ABB RobotStudio station: RobotStudio-Project-01.rspag

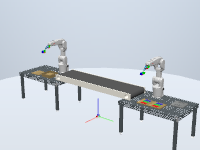
--- station ---
Station RobotStudio-Project-01 (saved by RobotStudio 20.4.9280.0)
Controller Controller1, task T_ROB2: task frame (RAPID world) sits at (-301.82, 1547.77, 837.1) mm in the station
Controller Controller1, task T_ROB1: task frame (RAPID world) sits at (-301.82, 1547.77, 837.1) mm in the station
Controller Controller1
  mechanical unit ROB_1: IRB1200_5_90_STD_03_1, 6 joints, base frame (0, 0, 0) mm
  mechanical unit ROB_2: IRB1200_5_90_STD_03_2, 6 joints, base frame (0, -3095.03, 0) mm
Layout (positions relative to the parent item):
  - WALL [part]
  - CONV_BELT [part] at (300.5, 959.08, 865.68) mm, rotated rx 90 ry 0 rz -90 deg
  - TABLE_1 [part] at (-6.2, -768.26, 800) mm, rotated rx 90 ry 0 rz 180 deg
  - TABLE_2 [part] at (-5.7, -4268.26, 800) mm, rotated rx 90 ry 0 rz 180 deg
  - TAB_1_ALL [part] at (184.19, 1489.88, 847.1) mm
  - TAB_2_ALL [part] at (184.19, 1790.38, 847.1) mm
  - TAB_3_HOME [part] at (-149.02, 2188.84, 854.6) mm
  - BOX [part] at (204.09, -1572.68, 882.1) mm, rotated rx 180 ry 0 rz 180 deg
  - BOX_COVER_ONBOX [part] at (204.09, -1572.68, 882.1) mm, rotated rx 180 ry 0 rz 180 deg
  - BOX_COVER_HOME [part] at (209.09, -2017.68, 802.1) mm, rotated rx 180 ry 0 rz 180 deg
  - TAB_1_POS_1 [part] at (184.19, 1489.88, 847.1) mm
  - TAB_1_POS_3 [part] at (184.19, 1489.88, 847.1) mm
  - TAB_1_POS_2 [part] at (184.19, 1489.88, 847.1) mm
  - TAB_2_POS_1 [part] at (184.19, 1790.38, 847.1) mm
  - TAB_2_POS_3 [part] at (184.19, 1790.38, 847.1) mm
  - TAB_2_POS_2 [part] at (184.19, 1790.38, 847.1) mm
  - TAB_3_CONV_1 [part] at (1.48, 950, 994.6) mm
  - TAB_3_CONV_2 [part] at (1.48, -975, 994.6) mm
  - TAB_3_INBOX [part] at (191.48, -1570.66, 884.6) mm
  - TAB_3_CONV_1_POS_1 [part] at (1.48, 950, 994.6) mm
  - TAB_3_CONV_1_POS_2 [part] at (1.48, 950, 994.6) mm
  - IRB1200_5_90_STD_03_1 [mechanism, from Robots\IRB1200_5_90_STD_03.rslib] at (-301.82, 1547.77, 837.1) mm; joint values [0, 0, 0, 0, 0.5236, 0] (rad or m)
  - IRB1200_5_90_STD_03_2 [mechanism, from Robots\IRB1200_5_90_STD_03.rslib] at (-301.82, -1547.27, 837.1) mm; joint values [0, 0, 0, 0, 0.5236, 0] (rad or m)
  - smc_gripper_1 [mechanism, from .rslib\smc_gripper.rslib] at (220.19, 1547.77, 1685.2) mm, rotated rx 180 ry 60 rz 180 deg
  - smc_gripper_2 [mechanism, from .rslib\smc_gripper.rslib] at (220.19, -1547.27, 1685.2) mm, rotated rx 180 ry 60 rz 180 deg
  - Detacher_T3_1 [smart component, from Components\Detacher.rslib]
      properties: Child=TAB_3_HOME; KeepPosition=true
  - Attacher_T3_1 [smart component, from Components\Attacher.rslib]
      properties: Parent=smc_gripper_1; Flange=0; Child=TAB_3_HOME; Mount=false; Offset=[0 0 0]; Orientation=[0 0 0]
  - Attacher_T1_P1 [smart component, from Components\Attacher.rslib]
      properties: Parent=smc_gripper_1; Flange=0; Child=TAB_1_POS_1; Mount=false; Offset=[0 0 0]; Orientation=[0 0 0]
  - Detacher_T1_P1 [smart component, from Components\Detacher.rslib]
      properties: Child=TAB_1_POS_1; KeepPosition=true
  - Attacher_T2_P1 [smart component, from Components\Attacher.rslib]
      properties: Parent=smc_gripper_1; Flange=0; Child=TAB_2_POS_1; Mount=false; Offset=[0 0 0]; Orientation=[0 0 0]
  - Detacher_T2_P1 [smart component, from Components\Detacher.rslib]
      properties: Child=TAB_2_POS_1; KeepPosition=true
  - Attacher_T1_P2 [smart component, from Components\Attacher.rslib]
      properties: Parent=smc_gripper_1; Flange=0; Child=TAB_1_POS_2; Mount=false; Offset=[0 0 0]; Orientation=[0 0 0]
  - Detacher_T1_P2 [smart component, from Components\Detacher.rslib]
      properties: Child=TAB_1_POS_2; KeepPosition=true
  - Attacher_T2_P2 [smart component, from Components\Attacher.rslib]
      properties: Parent=smc_gripper_1; Flange=0; Child=TAB_2_POS_2; Mount=false; Offset=[0 0 0]; Orientation=[0 0 0]
  - Detacher_T2_P2 [smart component, from Components\Detacher.rslib]
      properties: Child=TAB_2_POS_2; KeepPosition=true
  - Attacher_T1_P3 [smart component, from Components\Attacher.rslib]
      properties: Parent=smc_gripper_1; Flange=0; Child=TAB_1_POS_3; Mount=false; Offset=[0 0 0]; Orientation=[0 0 0]
  - Detacher_T1_P3 [smart component, from Components\Detacher.rslib]
      properties: Child=TAB_1_POS_3; KeepPosition=true
  - Attacher_T2_P3 [smart component, from Components\Attacher.rslib]
      properties: Parent=smc_gripper_1; Flange=0; Child=TAB_2_POS_3; Mount=false; Offset=[0 0 0]; Orientation=[0 0 0]
  - Detacher_T2_P3 [smart component, from Components\Detacher.rslib]
      properties: Child=TAB_2_POS_3; KeepPosition=true
  - Attacher_T3_2 [smart component, from Components\Attacher.rslib]
      properties: Parent=smc_gripper_2; Flange=0; Child=TAB_3_HOME; Mount=false; Offset=[0 0 0]; Orientation=[0 0 0]
  - Detacher_T3_2 [smart component, from Components\Detacher.rslib]
      properties: Child=TAB_3_HOME; KeepPosition=true
  - Attacher_BC [smart component, from Components\Attacher.rslib]
      properties: Parent=smc_gripper_2; Flange=0; Child=BOX_COVER_HOME; Mount=false; Offset=[0 0 0]; Orientation=[0 0 0]
  - Detacher_BC [smart component, from Components\Detacher.rslib]
      properties: Child=BOX_COVER_HOME; KeepPosition=true
  - Attacher_T3_T1_P1 [smart component, from Components\Attacher.rslib]
      properties: Parent=TAB_3_HOME; Flange=0; Child=TAB_1_POS_1; Mount=false; Offset=[0 0 0]; Orientation=[0 0 0]
  - Detacher_T3_T1_P1 [smart component, from Components\Detacher.rslib]
      properties: Child=TAB_1_POS_1; KeepPosition=true
  - Attacher_T3_T2_P1 [smart component, from Components\Attacher.rslib]
      properties: Parent=TAB_3_HOME; Flange=0; Child=TAB_2_POS_1; Mount=false; Offset=[0 0 0]; Orientation=[0 0 0]
  - Detacher_T3_T2_P1 [smart component, from Components\Detacher.rslib]
      properties: Child=TAB_2_POS_1; KeepPosition=true
  - Attacher_T3_T1_P2 [smart component, from Components\Attacher.rslib]
      properties: Parent=TAB_3_HOME; Flange=0; Child=TAB_1_POS_2; Mount=false; Offset=[0 0 0]; Orientation=[0 0 0]
  - Attacher_T3_T2_P2 [smart component, from Components\Attacher.rslib]
      properties: Parent=TAB_3_HOME; Flange=0; Child=TAB_2_POS_2; Mount=false; Offset=[0 0 0]; Orientation=[0 0 0]
  - Attacher_T3_T1_P3 [smart component, from Components\Attacher.rslib]
      properties: Parent=TAB_3_HOME; Flange=0; Child=TAB_1_POS_3; Mount=false; Offset=[0 0 0]; Orientation=[0 0 0]
  - Attacher_T3_T2_P3 [smart component, from Components\Attacher.rslib]
      properties: Parent=TAB_3_HOME; Flange=0; Child=TAB_2_POS_3; Mount=false; Offset=[0 0 0]; Orientation=[0 0 0]
  - Detacher_T3_T1_P2 [smart component, from Components\Detacher.rslib]
      properties: Child=TAB_1_POS_2; KeepPosition=true
  - Detacher_T3_T2_P2 [smart component, from Components\Detacher.rslib]
      properties: Child=TAB_2_POS_2; KeepPosition=true
  - Detacher_T3_T1_P3 [smart component, from Components\Detacher.rslib]
      properties: Child=TAB_1_POS_3; KeepPosition=true
  - Detacher_T3_T2_P3 [smart component, from Components\Detacher.rslib]
      properties: Child=TAB_2_POS_3; KeepPosition=true
  - Positioner_T3_HOME [smart component, from Components\Positioner.rslib]
      properties: Object=TAB_3_HOME; Position=[-0.149017 2.188837 0.854598]; Orientation=[0 0 0]; Reference=Global; ReferenceObject=(none)
  - Positioner_T1_P1 [smart component, from Components\Positioner.rslib]
      properties: Object=TAB_1_POS_1; Position=[0.184195 1.489875 0.847098]; Orientation=[0 0 0]; Reference=Global; ReferenceObject=(none)
  - Positioner_T2_P1 [smart component, from Components\Positioner.rslib]
      properties: Object=TAB_2_POS_1; Position=[0.184195 1.790375 0.847098]; Orientation=[0 0 0]; Reference=Global; ReferenceObject=(none)
  - Positioner_T1_P2 [smart component, from Components\Positioner.rslib]
      properties: Object=TAB_1_POS_2; Position=[0.184195 1.489875 0.847098]; Orientation=[0 0 0]; Reference=Global; ReferenceObject=(none)
  - Positioner_T2_P2 [smart component, from Components\Positioner.rslib]
      properties: Object=TAB_2_POS_2; Position=[0.184195 1.790375 0.847098]; Orientation=[0 0 0]; Reference=Global; ReferenceObject=(none)
  - Positioner_T1_P3 [smart component, from Components\Positioner.rslib]
      properties: Object=TAB_1_POS_3; Position=[0.184195 1.489875 0.847098]; Orientation=[0 0 0]; Reference=Global; ReferenceObject=(none)
  - Positioner_T2_P3 [smart component, from Components\Positioner.rslib]
      properties: Object=TAB_2_POS_3; Position=[0.184195 1.790375 0.847098]; Orientation=[0 0 0]; Reference=Global; ReferenceObject=(none)
  - Positioner_BC_HOME [smart component, from Components\Positioner.rslib]
      properties: Object=BOX_COVER_HOME; Position=[0.209094 -2.017683 0.802098]; Orientation=[3.14159265358979 0 3.14159265358979]; Reference=Global; ReferenceObject=(none)
  - LinearMover [smart component, from Components\LinearMover.rslib]
      properties: Object=TAB_3_HOME; Direction=[0 -0.001 0]; Speed=0.15; Reference=Global; ReferenceObject=(none)
  - PlaneSensor [smart component, from Components\PlaneSensor.rslib] at (-150, 0, 0) mm, rotated rx 90 ry 0 rz 0 deg
      properties: Origin=[0.0005 0.987098 1.113838]; Axis1=[0.3 0 0]; Axis2=[0 0.02 0]; SensedPart=(none)
    - _sensorPart_ [part]
  - LogicGate [smart component, from Components\LogicGate.rslib]
      properties: Operator=AND; Delay=0
  - LogicGate_2 [smart component, from Components\LogicGate.rslib]
      properties: Operator=NOT; Delay=0
Attachment: smc_gripper_1 is attached to IRB1200_5_90_STD_03_1 / Link6
Attachment: smc_gripper_2 is attached to IRB1200_5_90_STD_03_2 / Link6
Attachment: TAB_1_POS_2 is attached to TAB_3_HOME
Attachment: TAB_2_POS_2 is attached to TAB_3_HOME
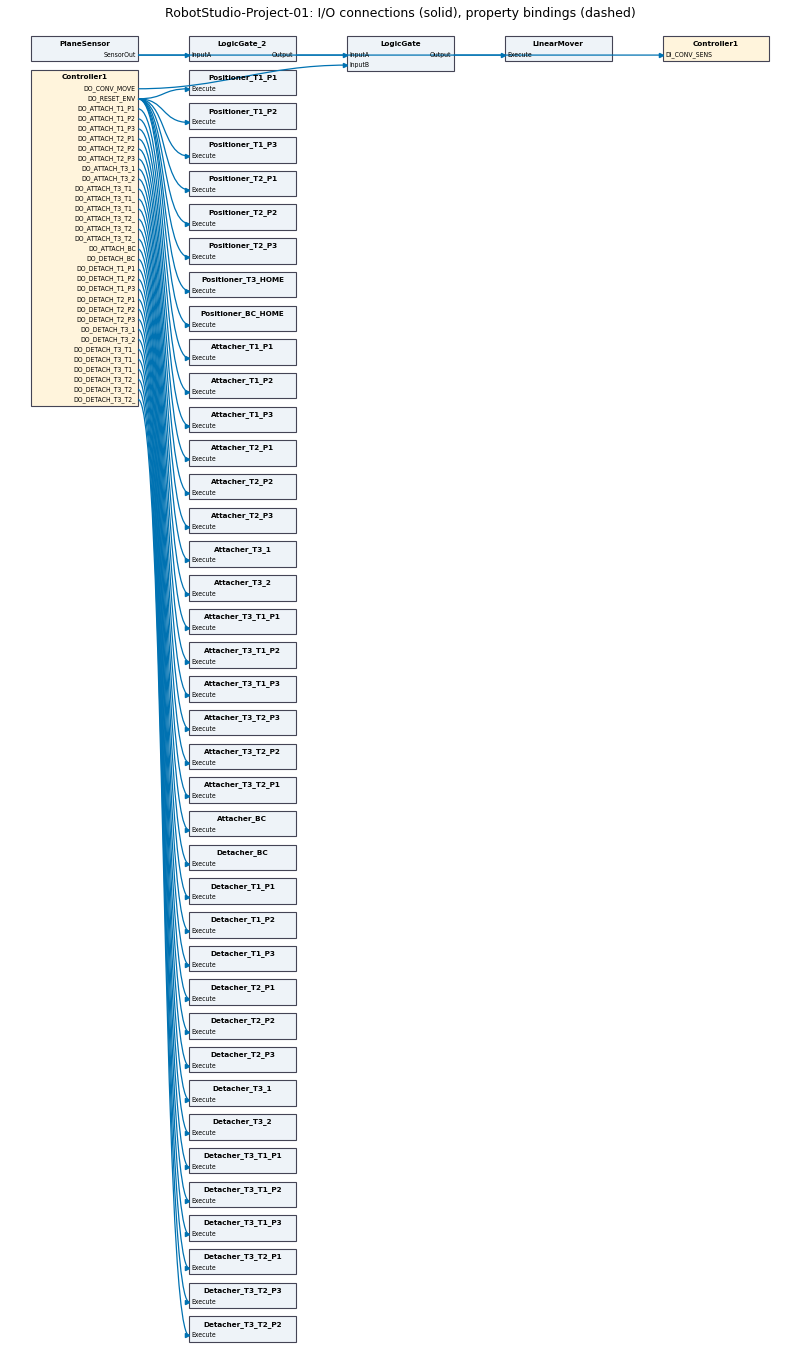
Station logic (signal -> signal, property => property):
  PlaneSensor.SensorOut -> Controller1.DI_CONV_SENS
  PlaneSensor.SensorOut -> LogicGate_2.InputA
  LogicGate_2.Output -> LogicGate.InputA
  Controller1.DO_CONV_MOVE -> LogicGate.InputB
  LogicGate.Output -> LinearMover.Execute
  Controller1.DO_RESET_ENV -> Positioner_T1_P1.Execute
  Controller1.DO_RESET_ENV -> Positioner_T1_P2.Execute
  Controller1.DO_RESET_ENV -> Positioner_T1_P3.Execute
  Controller1.DO_RESET_ENV -> Positioner_T2_P1.Execute
  Controller1.DO_RESET_ENV -> Positioner_T2_P2.Execute
  Controller1.DO_RESET_ENV -> Positioner_T2_P3.Execute
  Controller1.DO_RESET_ENV -> Positioner_T3_HOME.Execute
  Controller1.DO_RESET_ENV -> Positioner_BC_HOME.Execute
  Controller1.DO_ATTACH_T1_P1 -> Attacher_T1_P1.Execute
  Controller1.DO_ATTACH_T1_P2 -> Attacher_T1_P2.Execute
  Controller1.DO_ATTACH_T1_P3 -> Attacher_T1_P3.Execute
  Controller1.DO_ATTACH_T2_P1 -> Attacher_T2_P1.Execute
  Controller1.DO_ATTACH_T2_P2 -> Attacher_T2_P2.Execute
  Controller1.DO_ATTACH_T2_P3 -> Attacher_T2_P3.Execute
  Controller1.DO_ATTACH_T3_1 -> Attacher_T3_1.Execute
  Controller1.DO_ATTACH_T3_2 -> Attacher_T3_2.Execute
  Controller1.DO_ATTACH_T3_T1_P1 -> Attacher_T3_T1_P1.Execute
  Controller1.DO_ATTACH_T3_T1_P2 -> Attacher_T3_T1_P2.Execute
  Controller1.DO_ATTACH_T3_T1_P3 -> Attacher_T3_T1_P3.Execute
  Controller1.DO_ATTACH_T3_T2_P3 -> Attacher_T3_T2_P3.Execute
  Controller1.DO_ATTACH_T3_T2_P2 -> Attacher_T3_T2_P2.Execute
  Controller1.DO_ATTACH_T3_T2_P1 -> Attacher_T3_T2_P1.Execute
  Controller1.DO_ATTACH_BC -> Attacher_BC.Execute
  Controller1.DO_DETACH_BC -> Detacher_BC.Execute
  Controller1.DO_DETACH_T1_P1 -> Detacher_T1_P1.Execute
  Controller1.DO_DETACH_T1_P2 -> Detacher_T1_P2.Execute
  Controller1.DO_DETACH_T1_P3 -> Detacher_T1_P3.Execute
  Controller1.DO_DETACH_T2_P1 -> Detacher_T2_P1.Execute
  Controller1.DO_DETACH_T2_P2 -> Detacher_T2_P2.Execute
  Controller1.DO_DETACH_T2_P3 -> Detacher_T2_P3.Execute
  Controller1.DO_DETACH_T3_1 -> Detacher_T3_1.Execute
  Controller1.DO_DETACH_T3_2 -> Detacher_T3_2.Execute
  Controller1.DO_DETACH_T3_T1_P1 -> Detacher_T3_T1_P1.Execute
  Controller1.DO_DETACH_T3_T1_P2 -> Detacher_T3_T1_P2.Execute
  Controller1.DO_DETACH_T3_T1_P3 -> Detacher_T3_T1_P3.Execute
  Controller1.DO_DETACH_T3_T2_P1 -> Detacher_T3_T2_P1.Execute
  Controller1.DO_DETACH_T3_T2_P3 -> Detacher_T3_T2_P3.Execute
  Controller1.DO_DETACH_T3_T2_P2 -> Detacher_T3_T2_P2.Execute

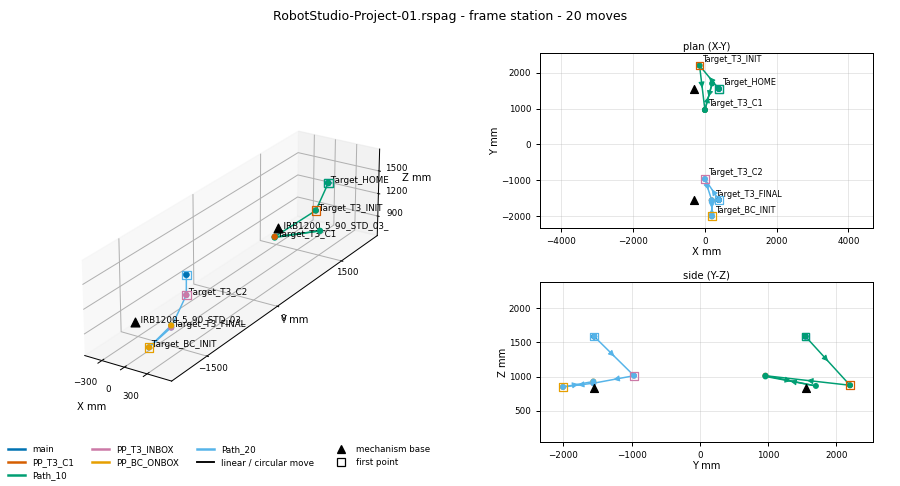
[picture p0: tool path of RobotStudio-Project-01.rspag in frame station, 20 of 38 moves have a stored position in this frame; points joined in program order, loops and branches not executed]
--- Backups/Controller1/RAPID/TASK1/PROGMOD/CalibData.mod ---
MODULE CalibData
    PERS tooldata smc_gripper:=[TRUE,[[0,0.004,197.001],[1,0,0,0]],[1,[0.207,-0.496,71.18],[1,0,0,0],0,0,0]];
ENDMODULE

--- Backups/Controller1/RAPID/TASK1/PROGMOD/Module1.mod ---
MODULE Module1

    ! Environment parameters structure
    RECORD environment_param_struct
        num T12_x_offset;
        num T12_y_offset;
        num T3_C1_x_offset;
    ENDRECORD

    ! Robot parameters structure
    RECORD robot_param_struct
        speeddata speed;
        zonedata zone;
        num object_z_offset;
    ENDRECORD

    ! Robot control structure
    RECORD robot_ctrl_struct
        num actual_state;
        num object_type;
        num tab_counter;
        robot_param_struct rob_par;
        environment_param_struct env_par;
    ENDRECORD

    ! Call main structure
    VAR robot_ctrl_struct rob_ctrl;

    ! Main waypoints (targets) for robot motion control
    CONST robtarget Target_HOME:=[[692.621953681,0.004,749.5995],[0.5,0,0.866025404,0],[0,-1,0,0],[9E+09,9E+09,9E+09,9E+09,9E+09,9E+09]];
    CONST robtarget Target_T3_INIT:=[[151.824,652.233,35],[0,0,1,0],[0,0,0,0],[9E+09,9E+09,9E+09,9E+09,9E+09,9E+09]];
    CONST robtarget Target_T3_C1:=[[302.324,-586.604,175],[0,0,1,0],[0,0,0,0],[9E+09,9E+09,9E+09,9E+09,9E+09,9E+09]];
    CONST robtarget Target_T12_P123:=[[502.324,152.483,25],[0,0,1,0],[0,0,0,0],[9E+09,9E+09,9E+09,9E+09,9E+09,9E+09]];
    CONST robtarget Target_T3_P12:=[[302.324,-586.604,164.256],[0,0,1,0],[0,0,0,0],[9E+09,9E+09,9E+09,9E+09,9E+09,9E+09]];

    ! ########################### ABB IRB 1200 (T_ROB1) MAIN CYCLE ########################### !
    PROC main()
        TEST rob_ctrl.actual_state
            CASE 0:
                ! *********************** INITIALIZATION STATE *********************** !
                ! Restore the environment
                RESET_ENV;
                ! Initialize the parameters
                INIT_PARAMS;
                ! Move -> home position
                MoveL Target_HOME,rob_ctrl.rob_par.speed,fine,smc_gripper\WObj:=wobj0;
                ! Change state -> {TRANSPORT OBJECT -> CONVEYOR BELT}
                rob_ctrl.actual_state := 1;
            CASE 1:
                ! *********************** P&P TAB_3 (TRANSPORT) OBJECT STATE *********************** !
                ! Pick the transport object and place it on the conveyor belt.
                PP_T3_C1;
                ! Change state -> {COLOR OBJECTS -> TRANSPORT OBJECT}
                rob_ctrl.actual_state := 2;
            CASE 2:
                ! *********************** P&P TAB_1_POS_A + TAB_2_POS_A (COLOR) OBJECTS STATE *********************** !
                ! Pick color objects and place them in the transport object (the color of the object is determined by the user).
                FOR i FROM 1 TO rob_ctrl.tab_counter DO
                    PP_T12_P123(i);
                ENDFOR
                ! Change state -> {BACK TO THE HOME}
                rob_ctrl.actual_state := 3;
            CASE 3:
                ! *********************** BACK TO THE HOME STATE *********************** !
                ! Move -> home position
                MoveL Target_HOME,rob_ctrl.rob_par.speed,fine,smc_gripper\WObj:=wobj0;
                ! Change state -> {START THE CONVEYOR BELT}
                rob_ctrl.actual_state := 4;
            CASE 4:
                ! *********************** START THE CONVEYOR BELT *********************** !
                ! Use the conveyor belt to move the transport object to the second robot.
                SetDO DO_CONV_MOVE, 1;
                ! Change state -> {EMPTY}
                rob_ctrl.actual_state := 5;
            CASE 5:
                ! *********************** EMPTY STATE *********************** !
        ENDTEST
    ENDPROC

    ! ########################### RESET ENVIRONMENT ########################### !
    PROC RESET_ENV()
        ! Detacher -> Robot No. 1
        PulseDO DO_DETACH_T1_P1;
        PulseDO DO_DETACH_T1_P2;
        PulseDO DO_DETACH_T1_P3;
        PulseDO DO_DETACH_T2_P1;
        PulseDO DO_DETACH_T2_P2;
        PulseDO DO_DETACH_T2_P3;
        PulseDO DO_DETACH_T3_1;
        ! Detacher -> Environment
        PulseDO DO_DETACH_T3_T1_P1;
        PulseDO DO_DETACH_T3_T1_P2;
        PulseDO DO_DETACH_T3_T1_P3;
        PulseDO DO_DETACH_T3_T2_P1;
        PulseDO DO_DETACH_T3_T2_P2;
        PulseDO DO_DETACH_T3_T2_P3;
        ! Restore position of the used objects
        PulseDO DO_RESET_ENV;
        ! Stop the Conveyor
        SetDO DO_CONV_MOVE, 0;
    ENDPROC

    ! ########################### INIT PARAMETERS ########################### !
    PROC INIT_PARAMS()
        ! Initialization the parameters of the robot
        ! Speed
        rob_ctrl.rob_par.speed := [800,800,800,800];
        ! Zone
        rob_ctrl.rob_par.zone := z50;
        ! Offset of the z-axis of the object
        rob_ctrl.rob_par.object_z_offset := 200;
        ! Object type -> 1 = POSITION 1 = RED; 2 = POSITION 2 = GREEN; 3 = POSITION 3 = BLUE;
        rob_ctrl.object_type := 2;
        ! The number of the color objects
        rob_ctrl.tab_counter := 2;
    ENDPROC

    ! ########################### P&P FUNCTION (TAB_3_HOME -> TAB_3_CONV_1) {TRANSPORT OBJECT -> CONVEYOR BELT} ########################### !
    PROC PP_T3_C1()
        ! ============= Pick trajectory ============= !
        MoveL Offs(Target_T3_INIT,0,0,rob_ctrl.rob_par.object_z_offset),rob_ctrl.rob_par.speed,rob_ctrl.rob_par.zone,smc_gripper\WObj:=wobj0;
        MoveL Offs(Target_T3_INIT,0,0,0),v200,fine,smc_gripper\WObj:=wobj0;
        WaitTime 0.25;
        ! Signal for the attacher
        PulseDO DO_ATTACH_T3_1;
        WaitTime 0.25;
        MoveL Offs(Target_T3_INIT,0,0,rob_ctrl.rob_par.object_z_offset),rob_ctrl.rob_par.speed,rob_ctrl.rob_par.zone,smc_gripper\WObj:=wobj0;
        MoveC Offs(Target_T12_P123,0,0,rob_ctrl.rob_par.object_z_offset), Offs(Target_T3_C1,0,0,rob_ctrl.rob_par.object_z_offset),rob_ctrl.rob_par.speed,rob_ctrl.rob_par.zone,smc_gripper\WObj:=wobj0;
        ! ============= Place trajectory ============= !
        MoveL Offs(Target_T3_C1,0,0,0),v200,fine,smc_gripper\WObj:=wobj0;
        WaitTime 0.25;
        ! Signal for the detacher
        PulseDO DO_DETACH_T3_1;
        WaitTime 0.25;
        MoveL Offs(Target_T3_C1,0,0,rob_ctrl.rob_par.object_z_offset),rob_ctrl.rob_par.speed,rob_ctrl.rob_par.zone,smc_gripper\WObj:=wobj0;
    ENDPROC

    ! ########################### P&P FUNCTION (TAB_1_POS_A + TAB_2_POS_A -> TAB_3_CONV_1_POS_B) {COLOR OBJECTS -> TRANSPORT OBJECT} ########################### !
    PROC PP_T12_P123(num tmp)
        ! Object type -> x-offset of the color objects
        ! Default x-coordinate of the target is in the center of the bins.
        IF rob_ctrl.object_type = 1 THEN
            rob_ctrl.env_par.T12_x_offset := 87.5;
        ELSEIF rob_ctrl.object_type = 2 THEN
            rob_ctrl.env_par.T12_x_offset := 0;
        ELSEIF rob_ctrl.object_type = 3 THEN
            rob_ctrl.env_par.T12_x_offset := -87.5;
        ENDIF
        ! The order of the object -> y-offset of the color object
        ! Default y-coordinate of the target is in the center of the bins.
        IF tmp = 1 THEN
            rob_ctrl.env_par.T12_y_offset := -150.25;
        ELSEIF tmp = 2 THEN
            rob_ctrl.env_par.T12_y_offset := 150.25;
        ENDIF
        ! ============= Pick trajectory ============= !
        MoveL Offs(Target_T12_P123,rob_ctrl.env_par.T12_x_offset,rob_ctrl.env_par.T12_y_offset,rob_ctrl.rob_par.object_z_offset),rob_ctrl.rob_par.speed,rob_ctrl.rob_par.zone,smc_gripper\WObj:=wobj0;
        MoveL Offs(Target_T12_P123,rob_ctrl.env_par.T12_x_offset,rob_ctrl.env_par.T12_y_offset,0),v200,fine,smc_gripper\WObj:=wobj0;
        WaitTime 0.25;
        ! The combination of the object type and its order -> signal for the attacher
        IF rob_ctrl.object_type = 1 THEN
            IF tmp = 1 THEN
                PulseDO DO_ATTACH_T1_P1;
            ELSEIF tmp = 2 THEN
                PulseDO DO_ATTACH_T2_P1;
            ENDIF
        ELSEIF rob_ctrl.object_type = 2 THEN
            IF tmp = 1 THEN
                PulseDO DO_ATTACH_T1_P2;
            ELSEIF tmp = 2 THEN
                PulseDO DO_ATTACH_T2_P2;
            ENDIF
        ELSEIF rob_ctrl.object_type = 3 THEN
            IF tmp = 1 THEN
                PulseDO DO_ATTACH_T1_P3;
            ELSEIF tmp = 2 THEN
                PulseDO DO_ATTACH_T2_P3;
            ENDIF
        ENDIF
        WaitTime 0.25;
        MoveL Offs(Target_T12_P123,rob_ctrl.env_par.T12_x_offset,rob_ctrl.env_par.T12_y_offset,rob_ctrl.rob_par.object_z_offset),rob_ctrl.rob_par.speed,rob_ctrl.rob_par.zone,smc_gripper\WObj:=wobj0;
        ! ============= Place trajectory ============= !
        ! The order of the object -> x-offset
        ! Default x-coordinate of the target is in the center of the TAB_3 (transport object) on the conveyor belt.
        IF tmp = 1 THEN
            rob_ctrl.env_par.T3_C1_x_offset := 87.5;
        ELSEIF tmp = 2 THEN
            rob_ctrl.env_par.T3_C1_x_offset := -87.5;
        ENDIF
        MoveL Offs(Target_T3_P12,rob_ctrl.env_par.T3_C1_x_offset,0,rob_ctrl.rob_par.object_z_offset),rob_ctrl.rob_par.speed,rob_ctrl.rob_par.zone,smc_gripper\WObj:=wobj0;
        MoveL Offs(Target_T3_P12,rob_ctrl.env_par.T3_C1_x_offset,0,0),v200,fine,smc_gripper\WObj:=wobj0;
        WaitTime 0.25;
        ! The combination of the object type and its order -> signal for the detacher
        ! Attach the color object to the TAB_3 (transport object) -> simulation logic
        IF rob_ctrl.object_type = 1 THEN
            IF tmp = 1 THEN
                PulseDO DO_DETACH_T1_P1;
                PulseDO DO_ATTACH_T3_T1_P1;
            ELSEIF tmp = 2 THEN
                PulseDO DO_DETACH_T2_P1;
                PulseDO DO_ATTACH_T3_T2_P1;
            ENDIF
        ELSEIF rob_ctrl.object_type = 2 THEN
            IF tmp = 1 THEN
                PulseDO DO_DETACH_T1_P2;
                PulseDO DO_ATTACH_T3_T1_P2;
            ELSEIF tmp = 2 THEN
                PulseDO DO_DETACH_T2_P2;
                PulseDO DO_ATTACH_T3_T2_P2;
            ENDIF
        ELSEIF rob_ctrl.object_type = 3 THEN
            IF tmp = 1 THEN
                PulseDO DO_DETACH_T1_P3;
                PulseDO DO_ATTACH_T3_T1_P3;
            ELSEIF tmp = 2 THEN
                PulseDO DO_DETACH_T2_P3;
                PulseDO DO_ATTACH_T3_T2_P3;
            ENDIF
        ENDIF
        WaitTime 0.25;
        MoveL Offs(Target_T3_P12,rob_ctrl.env_par.T3_C1_x_offset,0,rob_ctrl.rob_par.object_z_offset),rob_ctrl.rob_par.speed,rob_ctrl.rob_par.zone,smc_gripper\WObj:=wobj0;
    ENDPROC

    ! ########################### TEST TARGETS ########################### !
    PROC Path_10()
        MoveL Target_HOME,v800,fine,smc_gripper\WObj:=wobj0;
        MoveL Target_T3_INIT,v800,fine,smc_gripper\WObj:=wobj0;
        MoveL Target_T3_C1,v800,fine,smc_gripper\WObj:=wobj0;
        MoveL Target_T12_P123,v800,fine,smc_gripper\WObj:=wobj0;
        MoveL Target_T3_P12,v800,fine,smc_gripper\WObj:=wobj0;
    ENDPROC
ENDMODULE

--- Backups/Controller1/RAPID/TASK2/PROGMOD/Module1.mod ---
MODULE Module1

    ! Robot parameters structure
     RECORD robot_param_struct
        speeddata speed;
        zonedata zone;
        num object_z_offset;
    ENDRECORD

    ! Robot control structure
    RECORD robot_ctrl_struct
        num actual_state;
        robot_param_struct rob_par;
    ENDRECORD

    ! Call main structure
    VAR robot_ctrl_struct rob_ctrl;

    ! Main waypoints (targets) for robot motion control
    CONST robtarget Target_HOME:=[[692.621953681,-3095.03,749.5995],[0.5,0,0.866025404,0],[0,-1,0,0],[9E+09,9E+09,9E+09,9E+09,9E+09,9E+09]];
    CONST robtarget Target_T3_C2:=[[302.324,-2511.604,175],[0,0,1,0],[0,0,0,0],[9E+09,9E+09,9E+09,9E+09,9E+09,9E+09]];
    CONST robtarget Target_T3_FINAL:=[[492.324,-3107.267,65],[0,0,1,0],[0,0,0,0],[9E+09,9E+09,9E+09,9E+09,9E+09,9E+09]];
    CONST robtarget Target_BC_INIT:=[[497.324,-3552.267,10],[0,0,1,0],[0,0,0,0],[9E+09,9E+09,9E+09,9E+09,9E+09,9E+09]];
    CONST robtarget Target_BC_FINAL:=[[492.324,-3107.267,90],[0,0,1,0],[0,0,0,0],[9E+09,9E+09,9E+09,9E+09,9E+09,9E+09]];

    ! ########################### ABB IRB 1200 (T_ROB2) MAIN CYCLE ########################### !
    PROC main()
        TEST rob_ctrl.actual_state
            CASE 0:
                ! *********************** INITIALIZATION STATE *********************** !
                ! Restore the environment
                RESET_ENV;
                ! Initialize the parameters
                INIT_PARAMS;
                ! Move -> home position
                MoveL Target_HOME,rob_ctrl.rob_par.speed,fine,smc_gripper\WObj:=wobj0;
                ! Change state -> {STOP THE CONVEYOR BELT}
                rob_ctrl.actual_state := 1;
            CASE 1:
                ! *********************** STOP THE CONVEYOR BELT *********************** !
                ! Digital input -> conveyor sensor -> is the transport object in the position?
                IF DI_CONV_SENS = 1 THEN
                    SetDO DO_CONV_MOVE, 0;
                    ! Change state -> {TRANSPORT OBJECT -> IN THE BOX}
                    rob_ctrl.actual_state := 2;
                ENDIF
            CASE 2:
                ! *********************** P&P TAB_3 (TRANSPORT) OBJECT STATE *********************** !
                ! Pick the transport object and place it in the shipping box
                PP_T3_INBOX;
                ! Change state -> {BOX COVER -> ON THE BOX}
                rob_ctrl.actual_state := 3;
            CASE 3:
                ! *********************** P&P BOX COVER OBJECT STATE *********************** !
                ! Pick the box lid/cover and place it on the shipping box
                PP_BC_ONBOX;
                ! Change state -> {BACK TO THE HOME}
                rob_ctrl.actual_state := 4;
            CASE 4:
                ! *********************** BACK TO THE HOME STATE *********************** !
                ! Move -> home position
                MoveL Target_HOME,rob_ctrl.rob_par.speed,fine,smc_gripper\WObj:=wobj0;
                ! Change state -> {EMPTY}
                rob_ctrl.actual_state := 5;
            CASE 5:
                ! *********************** EMPTY STATE *********************** !
        ENDTEST
    ENDPROC

    ! ########################### RESET ENVIRONMENT ########################### !
    PROC RESET_ENV()
        ! Detacher -> Robot No. 2
        PulseDO DO_DETACH_T3_2;
        PulseDO DO_DETACH_BC;
        ! Restore position of the used objects
        PulseDO DO_RESET_ENV;
        ! Stop the Conveyor
        SetDO DO_CONV_MOVE, 0;
    ENDPROC

    ! ########################### INIT PARAMETERS ########################### !
    PROC INIT_PARAMS()
        ! Initialization the parameters of the robot
        ! Speed
        rob_ctrl.rob_par.speed := [800,800,800,800];
        ! Zone
        rob_ctrl.rob_par.zone := z50;
        ! Offset of the z-axis of the object
        rob_ctrl.rob_par.object_z_offset := 200;
    ENDPROC

    PROC PP_T3_INBOX()
        ! ============= Pick trajectory ============= !
        MoveL Offs(Target_T3_C2,0,0,rob_ctrl.rob_par.object_z_offset),rob_ctrl.rob_par.speed,rob_ctrl.rob_par.zone,smc_gripper\WObj:=wobj0;
        MoveL Offs(Target_T3_C2,0,0,0),v200,fine,smc_gripper\WObj:=wobj0;
        WaitTime 0.25;
        ! Signal for the attacher
        PulseDO DO_ATTACH_T3_2;
        WaitTime 0.25;
        MoveL Offs(Target_T3_C2,0,0,rob_ctrl.rob_par.object_z_offset),rob_ctrl.rob_par.speed,rob_ctrl.rob_par.zone,smc_gripper\WObj:=wobj0;
        ! ============= Place trajectory ============= !
        MoveL Offs(Target_T3_FINAL,0,0,rob_ctrl.rob_par.object_z_offset),rob_ctrl.rob_par.speed,rob_ctrl.rob_par.zone,smc_gripper\WObj:=wobj0;
        MoveL Offs(Target_T3_FINAL,0,0,0),v200,fine,smc_gripper\WObj:=wobj0;
        WaitTime 0.25;
        ! Signal for the detacher
        PulseDO DO_DETACH_T3_2;
        WaitTime 0.25;
        MoveL Offs(Target_T3_FINAL,0,0,rob_ctrl.rob_par.object_z_offset),rob_ctrl.rob_par.speed,rob_ctrl.rob_par.zone,smc_gripper\WObj:=wobj0;
    ENDPROC

    PROC PP_BC_ONBOX()
        ! ============= Pick trajectory ============= !
        MoveL Offs(Target_BC_INIT,0,0,rob_ctrl.rob_par.object_z_offset),rob_ctrl.rob_par.speed,rob_ctrl.rob_par.zone,smc_gripper\WObj:=wobj0;
        MoveL Offs(Target_BC_INIT,0,0,0),v200,fine,smc_gripper\WObj:=wobj0;
        WaitTime 0.25;
        ! Signal for the attacher
        PulseDO DO_ATTACH_BC;
        WaitTime 0.25;
        MoveL Offs(Target_BC_INIT,0,0,rob_ctrl.rob_par.object_z_offset),rob_ctrl.rob_par.speed,rob_ctrl.rob_par.zone,smc_gripper\WObj:=wobj0;
        ! ============= Place trajectory ============= !
        MoveL Offs(Target_BC_FINAL,0,0,rob_ctrl.rob_par.object_z_offset),rob_ctrl.rob_par.speed,rob_ctrl.rob_par.zone,smc_gripper\WObj:=wobj0;
        MoveL Offs(Target_BC_FINAL,0,0,0),v200,fine,smc_gripper\WObj:=wobj0;
        WaitTime 0.25;
        ! Signal for the detacher
        PulseDO DO_DETACH_BC;
        WaitTime 0.25;
        MoveL Offs(Target_BC_FINAL,0,0,rob_ctrl.rob_par.object_z_offset),rob_ctrl.rob_par.speed,rob_ctrl.rob_par.zone,smc_gripper\WObj:=wobj0;
    ENDPROC

    ! ########################### TEST TARGETS ########################### !
    PROC Path_20()
        MoveL Target_HOME,v800,fine,smc_gripper\WObj:=wobj0;
        MoveL Target_T3_C2,v800,fine,smc_gripper\WObj:=wobj0;
        MoveL Target_T3_FINAL,v800,fine,smc_gripper\WObj:=wobj0;
        MoveL Target_BC_INIT,v800,fine,smc_gripper\WObj:=wobj0;
        MoveL Target_BC_FINAL,v800,fine,smc_gripper\WObj:=wobj0;
    ENDPROC
ENDMODULE

--- Backups/Controller1/SYSPAR/EIO.cfg ---
EIO:CFG_1.0:6:1::
#
EIO_SIGNAL:

      -Name "DO_CONV_MOVE" -SignalType "DO"

      -Name "DI_CONV_SENS" -SignalType "DI"

      -Name "DO_RESET_ENV" -SignalType "DO"

      -Name "DO_ATTACH_T1_P1" -SignalType "DO"

      -Name "DO_ATTACH_T1_P2" -SignalType "DO"

      -Name "DO_ATTACH_T1_P3" -SignalType "DO"

      -Name "DO_ATTACH_T2_P1" -SignalType "DO"

      -Name "DO_ATTACH_T2_P2" -SignalType "DO"

      -Name "DO_ATTACH_T2_P3" -SignalType "DO"

      -Name "DO_ATTACH_T3_1" -SignalType "DO"

      -Name "DO_ATTACH_T3_2" -SignalType "DO"

      -Name "DO_ATTACH_T3_T1_P1" -SignalType "DO"

      -Name "DO_ATTACH_T3_T1_P2" -SignalType "DO"

      -Name "DO_ATTACH_T3_T1_P3" -SignalType "DO"

      -Name "DO_ATTACH_T3_T2_P3" -SignalType "DO"

      -Name "DO_ATTACH_T3_T2_P2" -SignalType "DO"

      -Name "DO_ATTACH_T3_T2_P1" -SignalType "DO"

      -Name "DO_ATTACH_BC" -SignalType "DO"

      -Name "DO_DETACH_BC" -SignalType "DO"

      -Name "DO_DETACH_T1_P1" -SignalType "DO"

      -Name "DO_DETACH_T1_P2" -SignalType "DO"

      -Name "DO_DETACH_T1_P3" -SignalType "DO"

      -Name "DO_DETACH_T2_P1" -SignalType "DO"

      -Name "DO_DETACH_T2_P2" -SignalType "DO"

      -Name "DO_DETACH_T2_P3" -SignalType "DO"

      -Name "DO_DETACH_T3_1" -SignalType "DO"

      -Name "DO_DETACH_T3_2" -SignalType "DO"

      -Name "DO_DETACH_T3_T1_P1" -SignalType "DO"

      -Name "DO_DETACH_T3_T1_P2" -SignalType "DO"

      -Name "DO_DETACH_T3_T1_P3" -SignalType "DO"

      -Name "DO_DETACH_T3_T2_P1" -SignalType "DO"

      -Name "DO_DETACH_T3_T2_P3" -SignalType "DO"

      -Name "DO_DETACH_T3_T2_P2" -SignalType "DO"
